// TwinCAT 3 PLC project ZaliczenieCwiczen
// ProgramVersion: 3.1.4023.0
// libraries:
//   Tc2_Standard, * (Beckhoff Automation GmbH)
//   Tc2_System, * (Beckhoff Automation GmbH)
//   Tc3_Module, * (Beckhoff Automation GmbH)
//   VisuDialogs, * (System)
//   VisuSymbols,3.5.10.0,System
// project tree:
//   DUTs/ E_kierunek.TcDUT, S_Macierz.TcDUT
//   / GlobalTextList.TcGTLO, PlcTask.TcTTO, Visualization Manager.TcVMO (not stored)
//   GVLs/ GVL_Lista.TcGVL
//   POUs/ Diagram Klas.TcCD (not stored), FB_Glowny.TcPOU, FB_Snake.TcPOU, MAIN.TcPOU
//   VISUs/ EkranGlowny.TcVIS, Snake.TcVIS
// real-time tasks:
//   TASK PlcTask: cycle T#10ms, priority 20, ADS port 350

CONFIGURATION ZaliczenieCwiczen
    RESOURCE PLC ON TwinCAT3
        TASK PlcTask(INTERVAL := T#10ms, PRIORITY := 20);
        PROGRAM MAIN WITH PlcTask : MAIN;
    END_RESOURCE
END_CONFIGURATION

// ---- DUTs/E_kierunek.TcDUT
{attribute 'qualified_only'}
{attribute 'strict'}
TYPE E_kierunek :
(
	lewo:=1,
	dol,
	prawo,
	gora
);
END_TYPE

// ---- DUTs/S_Macierz.TcDUT
TYPE S_Macierz :
STRUCT
	
	MacierzPola:ARRAY[1..10] OF ARRAY[1..10] OF BOOL;
	
END_STRUCT
END_TYPE

// ---- GVLs/GVL_Lista.TcGVL
{attribute 'qualified_only'}
VAR_GLOBAL
	
	iNajWynik:INT;
	iObecnyWynik:INT;
	bStanGry:BOOL;
	bStanStrzalek:ARRAY[1..4]OF BOOL; //prawa[1],dol[2],lewo[3],gora[4]
	bStanPrzyciskuRestart:BOOL;
	bStanPRzyciskuStartu:BOOL;
	iRekord:INT;
	
END_VAR

// ---- POUs/MAIN.TcPOU
PROGRAM MAIN
VAR
	ObranPoczatkowy:FB_Glowny;
	gra:FB_Snake;
END_VAR

ObranPoczatkowy();
gra();

END_PROGRAM

// ---- POUs/FB_Glowny.TcPOU
FUNCTION_BLOCK FB_Glowny
VAR
	iRuchX:INT:=50;
	iRuchY:INT:=50;
	predkoscRuchu:TIME:=T#2MS;
	czasoOdmierzacz:TON;
	timerRuchu:TON;
	iStan: INT;
END_VAR

CASE iStan OF
	
0:
	czasoOdmierzacz(IN:=TRUE, PT:=(predkoscRuchu/100));
	IF czasoOdmierzacz.Q=TRUE THEN
		iRuchY:=iRuchY+1;
		czasoOdmierzacz(IN:=FALSE);
	END_IF
	IF iRuchY=600 THEN
		iStan:=1;
	END_IF

1:
	czasoOdmierzacz(IN:=TRUE, PT:=(predkoscRuchu/100));
	IF czasoOdmierzacz.Q=TRUE THEN
		iRuchX:=iRuchX+1;
		czasoOdmierzacz(IN:=FALSE);
	END_IF
	IF iRuchX=1100 THEN
		iStan:=2;
	END_IF

2:
	czasoOdmierzacz(IN:=TRUE, PT:=(predkoscRuchu/100));
	IF czasoOdmierzacz.Q=TRUE THEN
		iRuchY:=iRuchY-1;
		czasoOdmierzacz(IN:=FALSE);
	END_IF
	IF iRuchY=50 THEN
		iStan:=3;
	END_IF


3:
	czasoOdmierzacz(IN:=TRUE, PT:=(predkoscRuchu/100));
	IF czasoOdmierzacz.Q=TRUE THEN
		iRuchX:=iRuchX-1;
		czasoOdmierzacz(IN:=FALSE);
	END_IF
	IF iRuchX=50 THEN
		iStan:=0;
	END_IF


END_CASE

END_FUNCTION_BLOCK

// ---- POUs/FB_Snake.TcPOU
FUNCTION_BLOCK FB_Snake EXTENDS FB_Glowny
VAR

	poleGry:S_Macierz;	
	
	wiersz:INT;//potem usunąć oba
	kolumna:INT;
	
	stanGry:INT:=3;

	iLicznikPrendkosci: INT;

	
	GAMEOVER:BOOL:=TRUE;
	EKRANSTARTOWY:BOOL:=FALSE;
	
	kierunek: INT;
	iLicznikKierunku: INT;
	kierunekRuchu:E_kierunek;
	
	stanJedzenia:BOOL;
	jedzeniePozycjaX:INT;
	jedzeniePozycjaY:INT;
	
	iLicnikPunktow:INT:=1;
	
	iWektorOgonaX:ARRAY[2..400] OF INT;
	iWektorOgonaY:ARRAY[2..400] OF INT;
	iLicznikY:INT:=2;

END_VAR

CASE stanGry OF
	
0:	
	FOR iLicznikKierunku:=1 TO 4  DO
		IF GVL_Lista.bStanStrzalek[iLicznikKierunku]=TRUE THEN
			kierunek:=iLicznikKierunku;							//sprawdzanie obecnego kierunku ruchu
			IF kierunek=1 THEN
				kierunekRuchu:=1;
			END_IF
			IF kierunek=2 THEN
				kierunekRuchu:=2;
			END_IF
			IF kierunek=3 THEN
				kierunekRuchu:=3;
			END_IF
			IF kierunek=4 THEN
				kierunekRuchu:=4;
			END_IF
		END_IF
	END_FOR
	M_SprawdzanieKolizji();
	IF stanJedzenia=FALSE THEN									//jeśli zdobędziemy punkt generuje nowe do zdobycia
		M_GenerowanieJedzenia();
	END_IF
	
	SUPER^.timerRuchu(IN:=TRUE,PT:=INT_TO_TIME(1000-(iLicznikPrendkosci*iLicnikPunktow))); //czas pomiędzy kolejnymi rychami 
	IF timerRuchu.Q=TRUE THEN
		IF  kierunek=1 THEN						//lewo
			iLicznikY:=iLicznikY+1;
			iWektorOgonaX[iLicznikY]:=wiersz;
			iWektorOgonaY[iLicznikY]:=kolumna;
			wiersz:=wiersz-1;
		END_IF
		
		IF  kierunek=2 THEN						//dół
			iLicznikY:=iLicznikY+1;
			iWektorOgonaX[iLicznikY]:=wiersz;
			iWektorOgonaY[iLicznikY]:=kolumna;
			kolumna:=kolumna+1;
			
		END_IF
		
		IF  kierunek=3 THEN						//prawo
			iLicznikY:=iLicznikY+1;
			iWektorOgonaX[iLicznikY]:=wiersz;
			iWektorOgonaY[iLicznikY]:=kolumna;
			wiersz:=wiersz+1;
			
		END_IF
		
		IF  kierunek=4 THEN						//góra
			iLicznikY:=iLicznikY+1;
			iWektorOgonaX[iLicznikY]:=wiersz;
			iWektorOgonaY[iLicznikY]:=kolumna;
			kolumna:=kolumna-1;
			
		END_IF
		
		stanGry:=1;
		
		IF kolumna>10 OR wiersz>10 OR kolumna<1 OR wiersz<1 THEN	// detekcja kolizji z ścianą
		stanGry:=2;
		END_IF
	END_IF

1:
	poleGry.MacierzPola[kolumna][wiersz]:=TRUE;
	timerRuchu(IN:=FALSE);
	M_Ogon();
	
	IF timerRuchu.Q=FALSE THEN
		IF iLicznikPrendkosci<100 THEN
			iLicznikPrendkosci:=iLicznikPrendkosci+1;
		END_IF
		IF jedzeniePozycjaX=wiersz AND jedzeniePozycjaY=kolumna THEN
			stanJedzenia:=FALSE;
			iLicnikPunktow:=iLicnikPunktow+1;
		END_IF
		stanGry:=0;
	END_IF
	
	
2:	
	M_NowaGra();

3:
	IF GVL_Lista.bStanPRzyciskuStartu=TRUE THEN
		M_Start();
	END_IF
END_CASE

METHOD M_GenerowanieJedzenia : BOOL
VAR
	iLicznik:INT;
END_VAR

jedzeniePozycjaX:=((iLicznikPrendkosci+wiersz) MOD 10)+1;	// z powodu iż w Twincacie nie mogłem znaleść funkcji RANDOM napisałem coś tkaiego, działa ale jest mało losowe
IF jedzeniePozycjaX <5 THEN
	jedzeniePozycjaX:=jedzeniePozycjaX + 2;
END_IF
jedzeniePozycjaY:=((jedzeniePozycjaX+kolumna) MOD 10)+1;
IF jedzeniePozycjaY<5 THEN
	jedzeniePozycjaY:=((jedzeniePozycjaY+wiersz) MOD 10)+1;
END_IF
IF jedzeniePozycjaX =wiersz OR jedzeniePozycjaY = kolumna THEN
	jedzeniePozycjaX:=((jedzeniePozycjaX+8) MOD 10)+1;
	jedzeniePozycjaY:=((jedzeniePozycjaX*jedzeniePozycjaY*iLicznikPrendkosci) MOD 10)+1; 
END_IF
poleGry.MacierzPola[jedzeniePozycjaY][jedzeniePozycjaX]:=TRUE;
StanJedzenia:=TRUE;
END_METHOD

METHOD M_NowaGra : BOOL
VAR
	i: INT;
	x: INT;
END_VAR
	poleGry.MacierzPola[jedzeniePozycjaY][jedzeniePozycjaX]:=FALSE;	
	GAMEOVER:=FALSE;													//wyłączenie informacji o przegranej grze
	IF iLicnikPunktow>GVL_Lista.iRekord THEN
		GVL_Lista.iRekord:=iLicnikPunktow;								// zapisanie liczby uzyskanych punktów
	END_IF
	FOR i:=1 TO 10 DO
		FOR x:=1 TO 10 DO
			poleGry.MacierzPola[x][i]:=FALSE;							// wyłączenie wszystkich pól
		END_FOR
	END_FOR
	IF GVL_Lista.bStanPrzyciskuRestart=TRUE THEN						//To samo co w przypadku metody M_Start
		THIS^.kolumna:=5;
		THIS^.wiersz:=6;
		THIS^.iWektorOgonaX[2]:=kolumna;
		THIS^.iWektorOgonaY[2]:=wiersz;
		THIS^.iLicznikY:=2;
		THIS^.kierunek:=0;
		THIS^.iLicnikPunktow:=1;
		THIS^.GAMEOVER:=TRUE;
		THIS^.iLicznikPrendkosci:=1;
		THIS^.stanJedzenia:=FALSE;
		THIS^.stanGry:=0;
	END_IF
END_METHOD

METHOD M_Ogon : BOOL
VAR
	//petla 1
	i:INT;
	x:INT;
	licznikOgona:INT;
	
	//liczenie co co skasowac
	q:INT;
	w:INT;
	
END_VAR
FOR i:=1 TO 10 DO
	FOR x:=1 TO 10 DO
		IF poleGry.MacierzPola[x][i]=TRUE THEN			
			licznikOgona:=licznikOgona+1;				//Pętal sprawdzająca czy długość = liczba punktów kiedy zdobędziemy punkt zwieksza długość
		END_IF
	END_FOR
END_FOR

IF (licznikOgona-1)>=iLicnikPunktow THEN
	q:=iWektorOgonaY[iLicznikY-(iLicnikPunktow-1)];	
	w:=iWektorOgonaX[iLicznikY-(iLicnikPunktow-1)];
	poleGry.MacierzPola[q][w]:=FALSE;					//usuwanie końca ogona
END_IF
END_METHOD

METHOD M_SprawdzanieKolizji : BOOL
VAR
	
	x:INT;
	
END_VAR
FOR x:=(iLicznikY-(iLicnikPunktow-1)) TO iLicznikY DO
	IF kierunek>0 THEN
			IF iWektorOgonaY[x]=kolumna AND iWektorOgonaX[x]=wiersz THEN	//jeżeli obecny stan kolumny i wierszu jest równy stanowi poprzedniemu -n to...
				stanGry:=2;													//to zmień stan gry
			END_IF
	END_IF
END_FOR
END_METHOD

METHOD M_Start : BOOL
VAR_INPUT
END_VAR
										//parametry zmiennych potrzebe przy starcie
	THIS^.kolumna:=6;  					//kolumna startowa
	THIS^.wiersz:=5;					//wiersz startowy
	THIS^.iWektorOgonaX[2]:=kolumna;	//macierz zapamiętujaca poprzednie stany
	THIS^.iWektorOgonaY[2]:=wiersz;
	THIS^.iLicznikPrendkosci:=1;		//restart prędkości
	THIS^.stanJedzenia:=FALSE;			//zmienna uruchamiająca proces tworzenia 'jedzenia dla wężyka'
	THIS^.EKRANSTARTOWY:=TRUE;			//wyłaczenie komunikatu
	THIS^.stanGry:=0;					//zmeina stanu programu
END_METHOD

END_FUNCTION_BLOCK

// ---- GlobalTextList.TcGTLO
TEXTLIST GlobalTextList
  735 = '%d'
  468 = '1'
  794 = '1.Przciski ruchu lepiej przytrzymywać !!!'
  231 = '1.Przciski ruchu lepiej przytrzymywać <1sekunde !!!'
  3 = '2.Teoretycznie powinno dać się sterować K.NUM'
  678 = '<'
  903 = '>'
  470 = 'kalendarz'
  104 = 'kalenddarz'
  273 = 'KONIEC GRY'
  137 = 'KONIEC GRY '
  917 = 'ms'
  121 = 'NACISNIJ START'
  713 = 'Nacisnij START'
  891 = 'Naciśnij START'
  586 = 'Najleprzy wynik %d'
  997 = 'Nalerzy kliknąć ikonkę żeby przejść dalej'
  439 = 'Obecny wynik'
  873 = 'Obecny wynik %d'
  474 = 'Obecny wynik: %d'
  570 = 'Przciski ruchu lepiej przytrzymywać !!!'
  499 = 'Prędkość opóżnienia ruchu'
  592 = 'Rekord: %d'
  814 = 'RESTART'
  938 = 'Snake'
  267 = 'START'
  150 = 'START ABY ZACZĄĆ'
  939 = 'v'
  495 = 'X'
  459 = 'XD'
  268 = '^'
END_TEXTLIST

// ---- VISUs/EkranGlowny.TcVIS
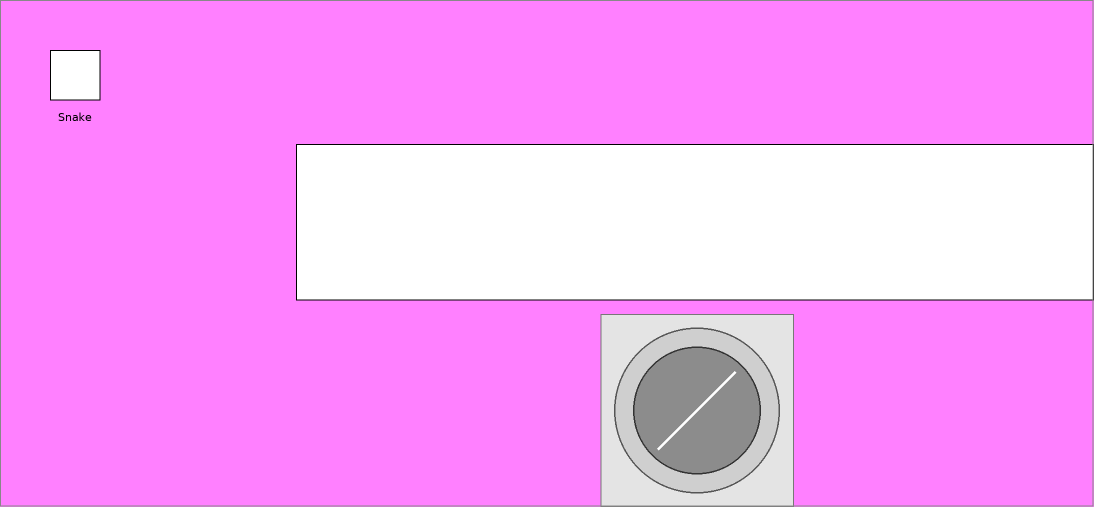
VISUALIZATION EkranGlowny  // 1094x507
    RoundedRectangle (50,50 50x50)
        p3560616238: MAIN.ObranPoczatkowy.iRuchX
        p2738717112: MAIN.ObranPoczatkowy.iRuchY
        OnMouseClick: change screen: Snake
    Rectangle (50,105 50x25), "Snake"
        p3560616238: MAIN.ObranPoczatkowy.iRuchX
        p2738717112: MAIN.ObranPoczatkowy.iRuchY
    Potentiometer360 (599,314 196x193), variable: MAIN.ObranPoczatkowy.predkoscRuchu, style: Potentiometer-Potentiometer360-Gray, scale format: %.1f, scale 1..111
        p2431819421: Outside
    RoundedRectangle (296,144 798x156), "Nalerzy kliknąć ikonkę żeby przejść dalej"
END_VISUALIZATION

// ---- VISUs/Snake.TcVIS
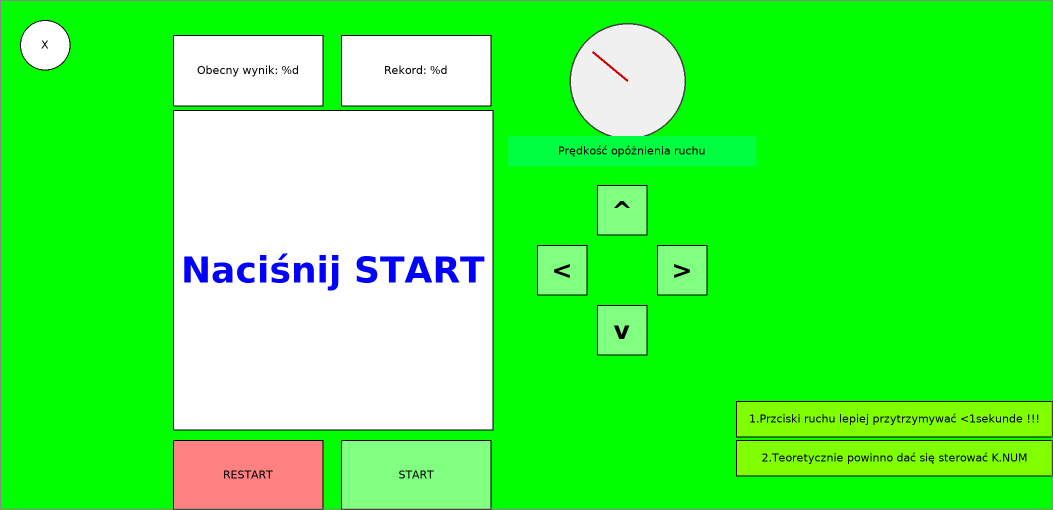
VISUALIZATION Snake  // 1053x510
    Rectangle (173,110 30x30), colour toggle: MAIN.gra.poleGry.MacierzPola[1][1]
    Rectangle (205,110 30x30), colour toggle: MAIN.gra.poleGry.MacierzPola[1][2]
    Rectangle (173,142 30x30), colour toggle: MAIN.gra.poleGry.MacierzPola[2][1]
    Rectangle (173,174 30x30), colour toggle: MAIN.gra.poleGry.MacierzPola[3][1]
    Rectangle (173,206 30x30), colour toggle: MAIN.gra.poleGry.MacierzPola[4][1]
    Rectangle (173,238 30x30), colour toggle: MAIN.gra.poleGry.MacierzPola[5][1]
    Rectangle (173,270 30x30), colour toggle: MAIN.gra.poleGry.MacierzPola[6][1]
    Rectangle (173,302 30x30), colour toggle: MAIN.gra.poleGry.MacierzPola[7][1]
    Rectangle (173,334 30x30), colour toggle: MAIN.gra.poleGry.MacierzPola[8][1]
    Rectangle (173,366 30x30), colour toggle: MAIN.gra.poleGry.MacierzPola[9][1]
    Rectangle (173,398 30x30), colour toggle: MAIN.gra.poleGry.MacierzPola[10][1]
    Rectangle (237,110 30x30), colour toggle: MAIN.gra.poleGry.MacierzPola[1][3]
    Rectangle (269,110 30x30), colour toggle: MAIN.gra.poleGry.MacierzPola[1][4]
    Rectangle (301,110 30x30), colour toggle: MAIN.gra.poleGry.MacierzPola[1][5]
    Rectangle (333,110 30x30), colour toggle: MAIN.gra.poleGry.MacierzPola[1][6]
    Rectangle (365,110 30x30), colour toggle: MAIN.gra.poleGry.MacierzPola[1][7]
    Rectangle (397,110 30x30), colour toggle: MAIN.gra.poleGry.MacierzPola[1][8]
    Rectangle (429,110 30x30), colour toggle: MAIN.gra.poleGry.MacierzPola[1][9]
    Rectangle (461,110 30x30), colour toggle: MAIN.gra.poleGry.MacierzPola[1][10]
    Rectangle (205,142 30x30), colour toggle: MAIN.gra.poleGry.MacierzPola[2][2]
    Rectangle (237,142 30x30), colour toggle: MAIN.gra.poleGry.MacierzPola[2][3]
    Rectangle (269,142 30x30), colour toggle: MAIN.gra.poleGry.MacierzPola[2][4]
    Rectangle (301,142 30x30), colour toggle: MAIN.gra.poleGry.MacierzPola[2][5]
    Rectangle (333,142 30x30), colour toggle: MAIN.gra.poleGry.MacierzPola[2][6]
    Rectangle (365,142 30x30), colour toggle: MAIN.gra.poleGry.MacierzPola[2][7]
    Rectangle (397,142 30x30), colour toggle: MAIN.gra.poleGry.MacierzPola[2][8]
    Rectangle (429,142 30x30), colour toggle: MAIN.gra.poleGry.MacierzPola[2][9]
    Rectangle (461,142 30x30), colour toggle: MAIN.gra.poleGry.MacierzPola[2][10]
    Rectangle (205,174 30x30), colour toggle: MAIN.gra.poleGry.MacierzPola[3][2]
    Rectangle (237,174 30x30), colour toggle: MAIN.gra.poleGry.MacierzPola[3][3]
    Rectangle (269,174 30x30), colour toggle: MAIN.gra.poleGry.MacierzPola[3][4]
    Rectangle (301,174 30x30), colour toggle: MAIN.gra.poleGry.MacierzPola[3][5]
    Rectangle (333,174 30x30), colour toggle: MAIN.gra.poleGry.MacierzPola[3][6]
    Rectangle (365,174 30x30), colour toggle: MAIN.gra.poleGry.MacierzPola[3][7]
    Rectangle (397,174 30x30), colour toggle: MAIN.gra.poleGry.MacierzPola[3][8]
    Rectangle (429,174 30x30), colour toggle: MAIN.gra.poleGry.MacierzPola[3][9]
    Rectangle (461,174 30x30), colour toggle: MAIN.gra.poleGry.MacierzPola[3][10]
    Rectangle (205,206 30x30), colour toggle: MAIN.gra.poleGry.MacierzPola[4][2]
    Rectangle (237,206 30x30), colour toggle: MAIN.gra.poleGry.MacierzPola[4][3]
    Rectangle (269,206 30x30), colour toggle: MAIN.gra.poleGry.MacierzPola[4][4]
    Rectangle (301,206 30x30), colour toggle: MAIN.gra.poleGry.MacierzPola[4][5]
    Rectangle (333,206 30x30), colour toggle: MAIN.gra.poleGry.MacierzPola[4][6]
    Rectangle (365,206 30x30), colour toggle: MAIN.gra.poleGry.MacierzPola[4][7]
    Rectangle (397,206 30x30), colour toggle: MAIN.gra.poleGry.MacierzPola[4][8]
    Rectangle (429,206 30x30), colour toggle: MAIN.gra.poleGry.MacierzPola[4][9]
    Rectangle (461,206 30x30), colour toggle: MAIN.gra.poleGry.MacierzPola[4][10]
    Rectangle (205,238 30x30), colour toggle: MAIN.gra.poleGry.MacierzPola[5][2]
    Rectangle (237,238 30x30), colour toggle: MAIN.gra.poleGry.MacierzPola[5][3]
    Rectangle (269,238 30x30), colour toggle: MAIN.gra.poleGry.MacierzPola[5][4]
    Rectangle (301,238 30x30), colour toggle: MAIN.gra.poleGry.MacierzPola[5][5]
    Rectangle (333,238 30x30), colour toggle: MAIN.gra.poleGry.MacierzPola[5][6]
    Rectangle (365,238 30x30), colour toggle: MAIN.gra.poleGry.MacierzPola[5][7]
    Rectangle (397,238 30x30), colour toggle: MAIN.gra.poleGry.MacierzPola[5][8]
    Rectangle (429,238 30x30), colour toggle: MAIN.gra.poleGry.MacierzPola[5][9]
    Rectangle (461,238 30x30), colour toggle: MAIN.gra.poleGry.MacierzPola[5][10]
    Rectangle (205,270 30x30), colour toggle: MAIN.gra.poleGry.MacierzPola[6][2]
    Rectangle (237,270 30x30), colour toggle: MAIN.gra.poleGry.MacierzPola[6][3]
    Rectangle (269,270 30x30), colour toggle: MAIN.gra.poleGry.MacierzPola[6][4]
    Rectangle (301,270 30x30), colour toggle: MAIN.gra.poleGry.MacierzPola[6][5]
    Rectangle (333,270 30x30), colour toggle: MAIN.gra.poleGry.MacierzPola[6][6]
    Rectangle (365,270 30x30), colour toggle: MAIN.gra.poleGry.MacierzPola[6][7]
    Rectangle (397,270 30x30), colour toggle: MAIN.gra.poleGry.MacierzPola[6][8]
    Rectangle (429,270 30x30), colour toggle: MAIN.gra.poleGry.MacierzPola[6][9]
    Rectangle (461,270 30x30), colour toggle: MAIN.gra.poleGry.MacierzPola[6][10]
    Rectangle (205,302 30x30), colour toggle: MAIN.gra.poleGry.MacierzPola[7][2]
    Rectangle (237,302 30x30), colour toggle: MAIN.gra.poleGry.MacierzPola[7][3]
    Rectangle (269,302 30x30), colour toggle: MAIN.gra.poleGry.MacierzPola[7][4]
    Rectangle (301,302 30x30), colour toggle: MAIN.gra.poleGry.MacierzPola[7][5]
    Rectangle (333,302 30x30), colour toggle: MAIN.gra.poleGry.MacierzPola[7][6]
    Rectangle (365,302 30x30), colour toggle: MAIN.gra.poleGry.MacierzPola[7][7]
    Rectangle (397,302 30x30), colour toggle: MAIN.gra.poleGry.MacierzPola[7][8]
    Rectangle (429,302 30x30), colour toggle: MAIN.gra.poleGry.MacierzPola[7][9]
    Rectangle (461,302 30x30), colour toggle: MAIN.gra.poleGry.MacierzPola[7][10]
    Rectangle (205,334 30x30), colour toggle: MAIN.gra.poleGry.MacierzPola[8][2]
    Rectangle (237,334 30x30), colour toggle: MAIN.gra.poleGry.MacierzPola[8][3]
    Rectangle (269,334 30x30), colour toggle: MAIN.gra.poleGry.MacierzPola[8][4]
    Rectangle (301,334 30x30), colour toggle: MAIN.gra.poleGry.MacierzPola[8][5]
    Rectangle (333,334 30x30), colour toggle: MAIN.gra.poleGry.MacierzPola[8][6]
    Rectangle (365,334 30x30), colour toggle: MAIN.gra.poleGry.MacierzPola[8][7]
    Rectangle (397,334 30x30), colour toggle: MAIN.gra.poleGry.MacierzPola[8][8]
    Rectangle (429,334 30x30), colour toggle: MAIN.gra.poleGry.MacierzPola[8][9]
    Rectangle (461,334 30x30), colour toggle: MAIN.gra.poleGry.MacierzPola[8][10]
    Rectangle (205,366 30x30), colour toggle: MAIN.gra.poleGry.MacierzPola[9][2]
    Rectangle (237,366 30x30), colour toggle: MAIN.gra.poleGry.MacierzPola[9][3]
    Rectangle (269,366 30x30), colour toggle: MAIN.gra.poleGry.MacierzPola[9][4]
    Rectangle (301,366 30x30), colour toggle: MAIN.gra.poleGry.MacierzPola[9][5]
    Rectangle (333,366 30x30), colour toggle: MAIN.gra.poleGry.MacierzPola[9][6]
    Rectangle (365,366 30x30), colour toggle: MAIN.gra.poleGry.MacierzPola[9][7]
    Rectangle (397,366 30x30), colour toggle: MAIN.gra.poleGry.MacierzPola[9][8]
    Rectangle (429,366 30x30), colour toggle: MAIN.gra.poleGry.MacierzPola[9][9]
    Rectangle (461,366 30x30), colour toggle: MAIN.gra.poleGry.MacierzPola[9][10]
    Rectangle (205,398 30x30), colour toggle: MAIN.gra.poleGry.MacierzPola[10][2]
    Rectangle (237,398 30x30), colour toggle: MAIN.gra.poleGry.MacierzPola[10][3]
    Rectangle (269,398 30x30), colour toggle: MAIN.gra.poleGry.MacierzPola[10][4]
    Rectangle (301,398 30x30), colour toggle: MAIN.gra.poleGry.MacierzPola[10][5]
    Rectangle (333,398 30x30), colour toggle: MAIN.gra.poleGry.MacierzPola[10][6]
    Rectangle (365,398 30x30), colour toggle: MAIN.gra.poleGry.MacierzPola[10][7]
    Rectangle (397,398 30x30), colour toggle: MAIN.gra.poleGry.MacierzPola[10][8]
    Rectangle (429,398 30x30), colour toggle: MAIN.gra.poleGry.MacierzPola[10][9]
    Rectangle (461,398 30x30), colour toggle: MAIN.gra.poleGry.MacierzPola[10][10]
    Ellipse (20,20 50x50), "X"
        OnMouseClick: change screen: EkranGlowny
    RoundedRectangle (173,440 150x70), "RESTART", colour toggle: GVL_Lista.bStanPrzyciskuRestart
        OnMouseDown: toggle GVL_Lista.bStanPrzyciskuRestart
        OnMouseUp: toggle GVL_Lista.bStanPrzyciskuRestart
    Rectangle (537,245 50x50), "<"
        OnMouseDown: toggle GVL_Lista.bStanStrzalek[1]
        OnMouseUp: toggle GVL_Lista.bStanStrzalek[1]
    Rectangle (597,305 50x50), "v"
        OnMouseDown: toggle GVL_Lista.bStanStrzalek[2]
        OnMouseUp: toggle GVL_Lista.bStanStrzalek[2]
    Rectangle (657,245 50x50), ">"
        OnMouseDown: toggle GVL_Lista.bStanStrzalek[3]
        OnMouseUp: toggle GVL_Lista.bStanStrzalek[3]
    Rectangle (597,185 50x50), "^"
        OnMouseDown: toggle GVL_Lista.bStanStrzalek[4]
        OnMouseUp: toggle GVL_Lista.bStanStrzalek[4]
    RoundedRectangle (173,35 150x71), "Obecny wynik: %d", text variable: MAIN.gra.iLicnikPunktow
    RoundedRectangle (341,35 150x71), "Rekord: %d", text variable: GVL_Lista.iRekord
    Rectangle (173,110 320x320), "KONIEC GRY", invisible if: MAIN.gra.GAMEOVER
    Rectangle (173,110 320x320), "Naciśnij START", invisible if: MAIN.gra.EKRANSTARTOWY
    RoundedRectangle (341,440 150x70), "START", colour toggle: GVL_Lista.bStanPRzyciskuStartu
        OnMouseDown: toggle GVL_Lista.bStanPRzyciskuStartu
        OnMouseUp: toggle GVL_Lista.bStanPRzyciskuStartu
    Meter180 (516,23 223x116), value: MAIN.gra.timerRuchu.PT, style: Meter-Meter180-Gray, scale format: %.1f, scale 0..1000
        p518627256: ms
    Rectangle (508,136 248x30), "Prędkość opóżnienia ruchu"
    Rectangle (736,401 317x36), "1.Przciski ruchu lepiej przytrzymywać <1sekunde !!!"
    Rectangle (736,440 317x36), "2.Teoretycznie powinno dać się sterować K.NUM"
    hotkey HotkeyInput Id=481047871488, Key=KeyDown=True, KeyName=8, VisuElemId=275
    hotkey HotkeyInput Id=481048920064, Key=KeyName=8, VisuElemId=275
    hotkey HotkeyInput Id=481049968640, Key=KeyDown=True, KeyName=4, VisuElemId=263
    hotkey HotkeyInput Id=481051017216, Key=KeyName=4, VisuElemId=263
    hotkey HotkeyInput Id=481052065792, Key=KeyDown=True, KeyName=6, VisuElemId=273
    hotkey HotkeyInput Id=481053114368, Key=KeyName=6, VisuElemId=273
    hotkey HotkeyInput Id=481054162944, Key=KeyDown=True, KeyName=2, VisuElemId=271
    hotkey HotkeyInput Id=481055211520, Key=KeyName=2, VisuElemId=271
END_VISUALIZATION
